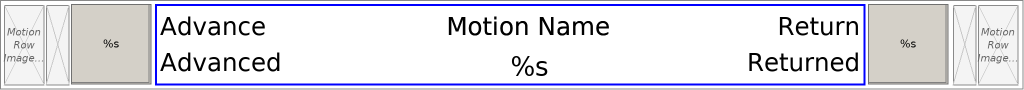
VISUALIZATION MotionRow  // 1024x90
VAR_IN_OUT
	MotionRowInstanceSingle:typeMotionRow; //feedback to motion row to operator
	MotionRowButtonsSingle:typeMotionRowButtons; //button feedback in seperate interface
END_VAR
    Rectangle (155,4 710x81)
    Button (868,4 80x80), "%s", text variable: MotionRowInstanceSingle.Returned.NumberOrder, invisible if: MotionRowInstanceSingle.Returned.bHideButton
        tap MotionRowButtonsSingle.btnReturn
    Button (71,4 80x80), "%s", text variable: MotionRowInstanceSingle.Advance.NumberOrder, invisible if: MotionRowInstanceSingle.Advance.bHideButton
        tap MotionRowButtonsSingle.btnAdvance
    Rectangle (393,50 273x33), "%s", text variable: MotionRowInstanceSingle.strPosn, invisible if: MotionRowInstanceSingle.bHidePosn
    Group (157,10 706x69)
        Rectangle (524,0 182x33), "Return", colour toggle: MotionRowInstanceSingle.Returned.RequestCoil, invisible if: MotionRowInstanceSingle.Returned.bHideCoil or MotionRowInstanceSingle.bIsAbsSymSwitch, text list: 'MotionRowText', text index: MotionRowInstanceSingle.IndexLocation + 3
        Rectangle (235,0 273x33), "Motion Name", invisible if: MotionRowInstanceSingle.bHideName or MotionRowInstanceSingle.bIsAbsSymSwitch, text list: 'MotionRowText', text index: MotionRowInstanceSingle.IndexLocation + 6
        Rectangle (524,36 182x33), "Returned", colour toggle: MotionRowInstanceSingle.Returned.Depth, invisible if: MotionRowInstanceSingle.Returned.bHideDepth or MotionRowInstanceSingle.bIsAbsSymSwitch, text list: 'MotionRowText', text index: MotionRowInstanceSingle.IndexLocation + 4
        Rectangle (0,0 207x33), "Advance", text variable: MotionRowInstanceSingle.Advance.valCoil, colour toggle: MotionRowInstanceSingle.Advance.RequestCoil, invisible if: MotionRowInstanceSingle.Advance.bHideCoil or MotionRowInstanceSingle.bIsAbsSymSwitch, text list: 'MotionRowText', text index: MotionRowInstanceSingle.IndexLocation + 0
        Rectangle (0,36 207x33), "Advanced", colour toggle: MotionRowInstanceSingle.Advance.Depth, invisible if: MotionRowInstanceSingle.Advance.bHideDepth or MotionRowInstanceSingle.bIsAbsSymSwitch, text list: 'MotionRowText', text index: MotionRowInstanceSingle.IndexLocation + 1
    Image (4,5 40x80), invisible if: NOT MotionRowInstanceSingle.Advance.InterlockOK OR MotionRowInstanceSingle.Advance.bHideInterlock, image: MotionRowImages.LeftHighlight
    Image (4,5 40x80), invisible if: MotionRowInstanceSingle.Advance.InterlockOK OR MotionRowInstanceSingle.Advance.bHideInterlock, image: MotionRowImages.LeftNot
    Image (978,5 40x80), invisible if: MotionRowInstanceSingle.Returned.InterlockOK OR MotionRowInstanceSingle.Returned.bHideInterlock, image: MotionRowImages.RightNot
    Image (978,5 40x80), invisible if: NOT MotionRowInstanceSingle.Returned.InterlockOK OR MotionRowInstanceSingle.Returned.bHideInterlock, image: MotionRowImages.RightHighlight
    Image (46,5 23x80), invisible if: MotionRowInstanceSingle.Advance.Prompt OR MotionRowInstanceSingle.Advance.bHidePrompt, image: MotionRowImages.PromptNOK
    Image (953,5 23x80), invisible if: NOT MotionRowInstanceSingle.Returned.Prompt OR MotionRowInstanceSingle.Returned.bHidePrompt, image: MotionRowImages.PromptOK
    Image (953,5 23x80), invisible if: MotionRowInstanceSingle.Returned.Prompt OR MotionRowInstanceSingle.Returned.bHidePrompt, image: MotionRowImages.PromptNOK
    Image (46,5 23x80), invisible if: NOT MotionRowInstanceSingle.Advance.Prompt OR MotionRowInstanceSingle.Advance.bHidePrompt, image: MotionRowImages.PromptOK
    Group (157,10 706x69)
        Rectangle (524,0 182x33), "Return", colour toggle: MotionRowInstanceSingle.Returned.RequestCoil, invisible if: MotionRowInstanceSingle.Returned.bHideCoil or NOT MotionRowInstanceSingle.bIsAbsSymSwitch, text list: 'MotionRowText', text index: MotionRowInstanceSingle.IndexLocation + 3 + 10
        Rectangle (235,0 273x33), "Motion Name", invisible if: MotionRowInstanceSingle.bHideName or NOT MotionRowInstanceSingle.bIsAbsSymSwitch, text list: 'MotionRowText', text index: MotionRowInstanceSingle.IndexLocation + 6 + 10
        Rectangle (524,36 182x33), "Returned", colour toggle: MotionRowInstanceSingle.Returned.Depth, invisible if: MotionRowInstanceSingle.Returned.bHideDepth or NOT MotionRowInstanceSingle.bIsAbsSymSwitch, text list: 'MotionRowText', text index: MotionRowInstanceSingle.IndexLocation + 4 + 10
        Rectangle (0,0 207x33), "Advance", text variable: MotionRowInstanceSingle.Advance.valCoil, colour toggle: MotionRowInstanceSingle.Advance.RequestCoil, invisible if: MotionRowInstanceSingle.Advance.bHideCoil or NOT MotionRowInstanceSingle.bIsAbsSymSwitch, text list: 'MotionRowText', text index: MotionRowInstanceSingle.IndexLocation + 0 + 10
        Rectangle (0,36 207x33), "Advanced", colour toggle: MotionRowInstanceSingle.Advance.Depth, invisible if: MotionRowInstanceSingle.Advance.bHideDepth or NOT MotionRowInstanceSingle.bIsAbsSymSwitch, text list: 'MotionRowText', text index: MotionRowInstanceSingle.IndexLocation + 1 + 10
END_VISUALIZATION

(* stored: Version 1.1.0.1, ProductVersion 3.1.4024.12
   Visu MotionRow: Id {23ea9bd1-da8d-4de5-b75e-eda7cd7af884} *)
